{attribute 'hide'}
{attribute 'reflection'}
FUNCTION_BLOCK TInteger
VAR
    Value : INT;
END_VAR

{attribute 'TcRpcEnable'}
METHOD Inc : INT
VAR_INPUT
END_VAR
Value := Value + 1;
Inc := Value;
END_METHOD

METHOD Init
VAR_INPUT
    Value : INT;
END_VAR
THIS^.Value := Value;
END_METHOD

END_FUNCTION_BLOCK

(* stored: Version 1.1.0.1, ProductVersion 3.1.4024.3
   POU TInteger: Id {686100c1-aadd-4e26-8abb-c08f1249a48a}, SpecialFunc None
   Method Inc: Id {466de744-80f3-4476-b5ef-d44705b51cdc}
   Method Init: Id {7d47b481-47d8-0f01-1201-274592ff66d6} *)
